FUNCTION_BLOCK UnitTestPrinterMock EXTENDS UnitTestPrinter
VAR_INPUT
END_VAR
VAR_OUTPUT
END_VAR
VAR
END_VAR

METHOD getFailMessage : MaxString
VAR_INPUT
END_VAR
getFailMessage := messageBuilder.toString();
END_METHOD

END_FUNCTION_BLOCK

(* stored: Version 1.1.0.1, ProductVersion 3.1.4022.12
   POU UnitTestPrinterMock: Id {7d78f928-4c3b-4ea2-a9f4-632deedb9e6f}, SpecialFunc None
   Method getFailMessage: Id {d91f44ec-251d-481d-998f-9e478b2a6031} *)
